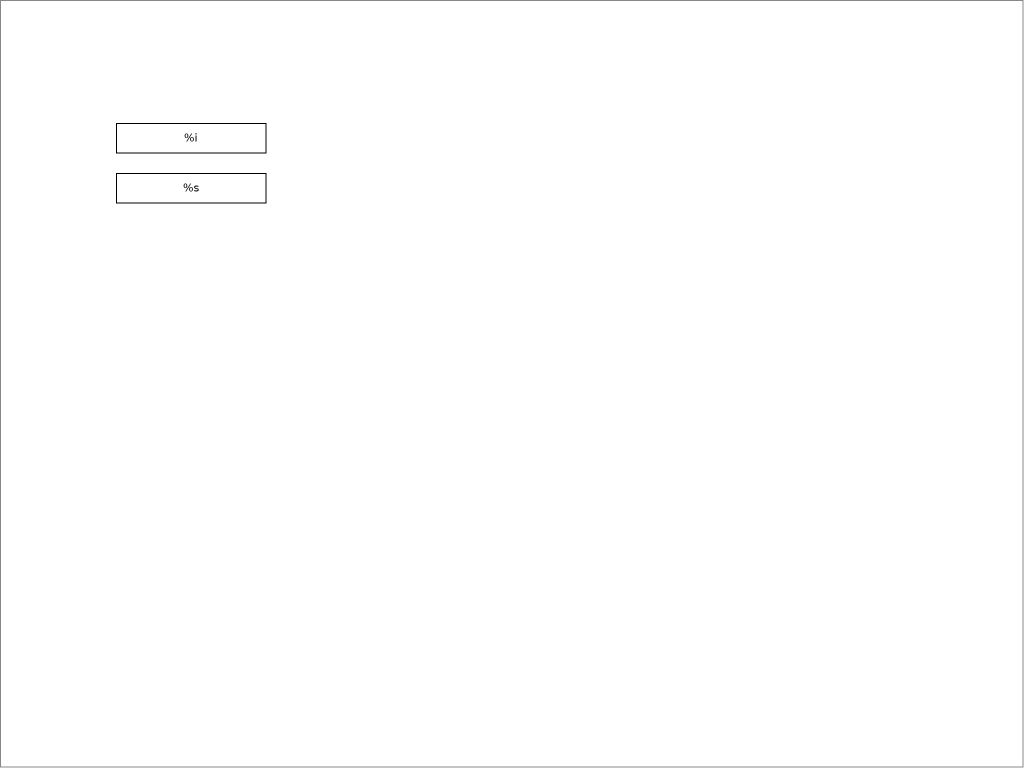
VISUALIZATION vMain  // 1024x768
    Rectangle (116,123 150x30), "%i", text variable: MAIN.nTest
        OnMouseDown: execute { gsPadTitle := 'Numpad nTest'; }
        OnMouseDown: write the text variable via Numpad
    Rectangle (116,173 150x30), "%s", text variable: MAIN.sTest
        OnMouseDown: execute { gsPadTitle := 'Keypad sTest'; }
        OnMouseDown: write the text variable via Keypad
END_VISUALIZATION

(* stored: Version 1.1.0.1, ProductVersion 3.1.4024.2
   Visu vMain: Id {a3394792-d1bf-4ce9-84a0-8f97cbaf968c} *)
